// TIA Portal V19 export
FUNCTION "FC_Takt_periodisch" : Void   // FC26, STL
{ S7_Optimized_Access := 'FALSE' }
// stored: AutoNumber false
   VAR_INPUT
      Freigabe : Bool;   // Taktung einschalten
      Timer_Nr : Timer;   // Timer für Takt
      Zeit_ein : S5Time;   // Einschaltzeit
      Zeit_aus : S5Time;   // Pausenzeit
   END_VAR
   VAR_OUTPUT
      on : Bool;   // Ausgang getaktet
   END_VAR
BEGIN

NETWORK
TITLE = Ausgang getaktet
      AN    #Freigabe;
      L     #Zeit_aus;
      SF    #Timer_Nr;

      A     #Freigabe;
      L     #Zeit_ein;
      SD    #Timer_Nr;

      AN    #Timer_Nr;
      A     #Freigabe;
      =     #on;

END_FUNCTION
